PROGRAM P_Demo_ConfirmAllAlarms
VAR
    fbLogger        : FB_TcEventLogger; // EventLogger 实例
    bConfirmAll     : BOOL := FALSE; // 上升沿触发
    bConfirmAllPrev : BOOL; // 边沿检测
    hr              : HRESULT; // 返回值监视
END_VAR

// =============================================================================
// 场景：管理员的「一键确认全部 WaitForConfirmation」操作
// 价值：一句调用完成批量确认
// 验证：操作前 HMI 有若干 WaitForConfirmation；写 bConfirmAll := TRUE 后全部变 Confirmed
// 验证步骤：
//   1. 右键 PLC 项目下 POUs 文件夹 → Add → Existing Item → 选本 .TcPOU 文件
//   2. 引用 Tc3_EventLogger（System → References → Add library）
//   3. 编译 → 登录 → 运行；按 verify 注释里给出的在线写值操作
// =============================================================================

IF bConfirmAll AND NOT bConfirmAllPrev THEN
    hr := fbLogger.ConfirmAllAlarms(nTimeStamp := 0);
END_IF;
bConfirmAllPrev := bConfirmAll;

END_PROGRAM

(* stored: Version 1.1.0.1, ProductVersion 3.1.4024.5
   POU P_Demo_ConfirmAllAlarms: Id {7485a2d1-f9d3-590e-911c-877feccb86b6}, SpecialFunc None *)
